// TwinCAT 3 PLC project PLC
// ProgramVersion: 3.1.4023.0
// libraries:
//   Tc2_Standard, * (Beckhoff Automation GmbH)
//   Tc2_System, * (Beckhoff Automation GmbH)
//   Tc2_Utilities, * (Beckhoff Automation GmbH)
//   Tc3_Module, * (Beckhoff Automation GmbH)
//   AX_Standard,1.24,Automate-X Ltd.
// project tree:
//   DUTs/Safety/ ST_Safety.TcDUT
//   GVLs/ GVL_EAP.TcGVL, GVL_HMI.TcGVL, GVL_IO.TcGVL, GVL_System.TcGVL, GVL_Recipe.TcGVL, GVL_Safety.TcGVL, GVL_Seq.TcGVL
//   / PlcTask.TcTTO
//   POUs/02 IO Mapping/ InputMapping.TcPOU, OutputMapping.TcPOU
//   POUs/03 Equipment/ DeviceInputs.TcPOU, DeviceOutputs.TcPOU
//   POUs/04 Program/ ExampleSequence.TcPOU
//   POUs/06 Safety/ Safety.TcPOU
//   POUs/09 General/ DataControl.TcPOU
//   POUs/10 EAP/ EAP_PublisherMapping.TcPOU, EAP_SubscriberMapping.TcPOU
//   POUs/ MachineStatePackML.TcPOU, MAIN.TcPOU
// real-time tasks:
//   TASK PlcTask: cycle T#10ms, priority 20, ADS port 350

CONFIGURATION PLC
    RESOURCE PLC ON TwinCAT3
        TASK PlcTask(INTERVAL := T#10ms, PRIORITY := 20);
        PROGRAM MAIN WITH PlcTask : MAIN;
    END_RESOURCE
END_CONFIGURATION

// ---- DUTs/Safety/ST_Safety.TcDUT
TYPE ST_Safety :
STRUCT
	

	//Basic Safety variables, add more if needed.
	bEStop					: BOOL;
	bEnergised				: BOOL;
	bHealthy				: BOOL;
	bEStopOk				: BOOL;
	bEStopResetRequired		: BOOL;
	

END_STRUCT
END_TYPE

// ---- GVLs/GVL_EAP.TcGVL
{attribute 'qualified_only'}

// Set size of array according to EAP data to be exchanged.

VAR_GLOBAL
	aPubBool		AT %Q*	: ARRAY [0..15] OF BOOL;		// EAP Published Array of Booleans
	aPubInt			AT %Q*	: ARRAY [0..15] OF INT;			// EAP Published Array of Integers
	aPubReal		AT %Q*	: ARRAY [0..15] OF REAL;		// EAP Published Array of Reals
	aSubBool		AT %I*	: ARRAY [0..15] OF BOOL;		// EAP Subscribed Array of Booleans
	aSubInt			AT %I*	: ARRAY [0..15] OF INT;			// EAP Subscribed Array of Integers
	aSubReal		AT %I*	: ARRAY [0..15] OF REAL;		// EAP Subscribed Array of Reals
END_VAR

// ---- GVLs/GVL_HMI.TcGVL
{attribute 'qualified_only'}
VAR_GLOBAL
END_VAR

// ---- GVLs/GVL_IO.TcGVL
{attribute 'qualified_only'}
VAR_GLOBAL
	

(* --- Digital Inputs --- *)


//Examples
//stPE3001				: ST_DigitalInput;
//stDI1001				: ST_DigitalInput;
//stPB4001				: ST_DigitalInput;
//stES4001				: ST_Safe2ChDigitalInput;		//PLC Cabinet Estop


(* --- Digital Outputs --- *)

//Examples
//stDO1001				: ST_DigitalOutput;		
//stDO1002				: ST_DigitalOutput;
//stSO4001				: ST_DigitalOutput;				//SO4001 Sounder


(* --- Analog Inputs --- *)

//Examples
//stAI4001				: ST_AnalogueInput;		
//stAI3001				: ST_AnalogueInput;



(* --- Analog Outputs --- *)

//Examples
//stAO4001				: ST_AnalogueInput;		
//stAO3001				: ST_AnalogueInput;



(* --- PLC IO Cards --- *)

//Examples
//stEL1008				: ST_EL1008; 
//stEL2008				: ST_EL2008;
//stEL3024				: ST_EL3024;

END_VAR

// ---- GVLs/GVL_System.TcGVL
{attribute 'qualified_only'}
VAR_GLOBAL
	
	MachineStates: ST_PackML;
	
	bResetSequenceTimerDefaults			: BOOL;				// Resets Sequence Timers to Defaults
	bSetDebounceTimes					: BOOL;				// Sets Photoeye Debounce Timers
	
END_VAR

// ---- GVLs/GVL_Recipe.TcGVL
{attribute 'qualified_only'}
VAR_GLOBAL
END_VAR

// ---- GVLs/GVL_Safety.TcGVL
{attribute 'qualified_only'}
VAR_GLOBAL
	

	stSafety			: ST_Safety;
	stSafetySeq			: ST_Sequence;
	fbSafetySeq			: FB_Sequence;
	
	bResetTrigger 		: BOOL; // from HMI or physical reset button

	bRun		AT %Q* 	: BOOL;	// To safety PLC
	bErrorAck   AT %Q* 	: BOOL;	// To safety PLC
	bReset    	AT %Q* 	: BOOL;	// To safety PLC
	
	bRunStatus  AT %I* 	: BOOL;	// From safety PLC
	
	bRequestToEnter		: BOOL; // Used with safety cages/doors
	
END_VAR

// ---- GVLs/GVL_Seq.TcGVL
{attribute 'qualified_only'}
VAR_GLOBAL
	
//List all sequencies 

//Example
//S101	 								: ST_Sequence;
//S102 									: ST_Sequence;

(* Exmaple Sequencies *)
stExampleSequence 						: ST_Sequence;
ExampleSequence_bHomingRequired 		: BOOL;

//Call  FB_Sequence for each sequence

//Example
//fbS101 								: FB_Sequence;
//fbS102 								: FB_Sequence;

(* Exmaple FB *)
fbExampleSequence : FB_Sequence;

// When used with conveyors , additions to Sequencies have been used on previous projects such as:
//S101_RequestingToSend		: BOOL;
//S101_ReadyToReceive       : BOOL; 

// When used with moving parts , additions to Sequencies have been used on previous projects such as:
//S101_bHomingRequired 		: BOOL;

END_VAR

// ---- POUs/MAIN.TcPOU
PROGRAM MAIN
VAR
END_VAR


// Add and Call Programs to be used 

//	InputMapping();
//	DeviceInputs();
//	Seq1();
//	Safety();
//	MachineStatePackML();
//	DataControl();
//	OutputMapping();
//	DeviceOutputs();
//	EAP_SubscriberMapping();
//	EAP_PublisherMapping();

END_PROGRAM

// ---- POUs/06 Safety/Safety.TcPOU
PROGRAM Safety
VAR
END_VAR


// Call Safety Sequence Function Block
GVL_Safety.fbSafetySeq(stSeq:=GVL_Safety.stSafetySeq);


CASE GVL_Safety.stSafetySeq.nStep OF
	0:	// Aborted
		// Actions
		
		
		// Step Transitions
		IF (GVL_Safety.bResetTrigger AND GVL_Safety.stSafetySeq.bStepTimerDn) THEN
			GVL_Safety.stSafetySeq.nNewStep := 1;
		END_IF
		
	1:	// Safety Reset Step 1
		// Actions
		
		// Step Transitions
		IF GVL_Safety.stSafetySeq.bStepTimerDn THEN
			GVL_Safety.stSafetySeq.nNewStep := 2;
		END_IF 
		
	2:	// Safety Reset Step 2
		// Actions

		// Step Transitions
		IF GVL_Safety.stSafetySeq.bStepTimerDn THEN
			GVL_Safety.stSafetySeq.nNewStep := 3;
		END_IF
		
	3:	// Safety Reset Step 3
		// Actions

		// Step Transitions
		IF GVL_Safety.stSafetySeq.bStepTimerDn AND GVL_Safety.stSafety.bHealthy THEN
			
			GVL_Safety.stSafetySeq.nNewStep := 4;
		END_IF 
		
	4: //System Reset Step 1
		// Actions
			
		// Step Transitions
		IF GVL_Safety.stSafetySeq.bStepTimerDn THEN
			GVL_Safety.stSafetySeq.nNewStep := 5;
		END_IF 

	5:	//System Reset Step 2
		// Actions

		// Step Transitions
		IF GVL_Safety.stSafetySeq.bStepTimerDn THEN
			GVL_Safety.stSafetySeq.nNewStep := 6;
		END_IF
		
	6: 	//System Reset Complete
		//Actions
		
		//Step Transitions

	
END_CASE

IF GVL_Safety.bResetTrigger THEN
	GVL_Safety.stSafetySeq.nNewStep := 1;
END_IF  

IF NOT GVL_Safety.stSafety.bHealthy THEN
	GVL_Safety.stSafetySeq.nNewStep := 0;
END_IF	

WriteToFlags();
WriteToOutputs();

ACTION WriteToFlags:




//Safety Group Run
IF 	GVL_Safety.stSafetySeq.nStep = 1 OR
	GVL_Safety.stSafetySeq.nStep = 2 OR
	GVL_Safety.stSafetySeq.nStep = 3 OR
	GVL_Safety.stSafetySeq.nStep = 4 OR
	GVL_Safety.stSafetySeq.nStep = 5 OR
	GVL_Safety.stSafetySeq.nStep = 6
THEN
	GVL_Safety.bRun := TRUE;
ELSE
	GVL_Safety.bRun := FALSE;
END_IF
		
//Safety Group Error Acknowledge Reset
IF 
	GVL_Safety.stSafetySeq.nStep = 2
THEN
	GVL_Safety.bErrorAck := TRUE;
ELSE
	GVL_Safety.bErrorAck := FALSE;
END_IF			
		

//Safety Function Block Resets
IF 
	GVL_Safety.stSafetySeq.nStep = 2
THEN
	GVL_Safety.bReset := TRUE;
ELSE
	GVL_Safety.bReset := FALSE;
END_IF
END_ACTION

ACTION WriteToOutputs:

END_ACTION

END_PROGRAM

// ---- POUs/02 IO Mapping/InputMapping.TcPOU
(*****************************************************************************************
	Automate-X Ltd. © 
	www.automate-x.nz 	
	
	Map Physical Inputs to device structures
******************************************************************************************)

PROGRAM InputMapping
VAR
END_VAR



// Map physical inputs (based on PLC IO Cards in GVL IO) to device structures
// This is IO Assignment based on PLC IO List in Equipment schedule



// This EXAMPLE is based on variables in GVL_IO

//EL1008 | 8-channel digital input terminal 24 V DC, 3 ms

//GVL_IO.stPE3001.bInput		:=  GVL_IO.stEL1008.bDI1;
//GVL_IO.stDI1001.bInput		:=  GVL_IO.stEL1008.bDI2;
//GVL_IO.stPB4001.bInput		:=  GVL_IO.stEL1008.bDI3;
// SPARE            		:=  GVL_IO.stEL1008.bDI4;
// SPARE            		:=  GVL_IO.stEL1008.bDI5;
// SPARE            		:=  GVL_IO.stEL1008.bDI6;
// SPARE            		:=  GVL_IO.stEL1008.bDI7;
// SPARE            		:=  GVL_IO.stEL1008.bDI8;



//EL3024 | 4-channel Analog Input terminal ,Current , 4..20mA, 12bit, Differential

//GVL_IO.stAO4001.bInput		:=  GVL_IO.stEL3024.bAI1;
//GVL_IO.stAO3001.bInput		:=  GVL_IO.stEL3024.bAI2;
// SPARE  					:=  GVL_IO.stEL3024.bAI3;
// SPARE            		:=  GVL_IO.stEL3024.bAI4;

END_PROGRAM

// ---- POUs/02 IO Mapping/OutputMapping.TcPOU
(*****************************************************************************************
	Automate-X Ltd. © 
	www.automate-x.nz 	
	
	Map Physical Outputs to device structures
******************************************************************************************)


PROGRAM OutputMapping
VAR
END_VAR




// Map physical inputs (based on PLC IO Cards in GVL IO) to device structures
// This is IO Assignment based on PLC IO List in Equipment schedule



// This EXAMPLE is based on variables in GVL_IO

//EL2008 | 8-channel digital Output terminal 24 V DC, 3 ms

//GVL_IO.stDO1001.bOutput		:=  GVL_IO.stEL2008.bDO1;
//GVL_IO.stDO1002.bOutput		:=  GVL_IO.stEL2008.bDO2;
//GVL_IO.stSO4001.bOutput		:=  GVL_IO.stEL2008.bDO3;
// SPARE            		:=  GVL_IO.stEL2008.bDO4;
// SPARE            		:=  GVL_IO.stEL2008.bDO5;
// SPARE            		:=  GVL_IO.stEL2008.bDO6;
// SPARE            		:=  GVL_IO.stEL2008.bDO7;
// SPARE            		:=  GVL_IO.stEL2008.bDO8;

END_PROGRAM

// ---- POUs/03 Equipment/DeviceInputs.TcPOU
(*****************************************************************************************
	Automate-X Ltd. ©  
	www.automate-x.nz 	
	
	Initialise and call all function blocks for Input type devices
******************************************************************************************)

PROGRAM DeviceInputs
VAR
	
//Example 
// fbPX01    	: FB_DigitalInput;
// fbDI1002		: FB_DigitalInput;		
// fbPE3001		: FB_DigitalInput;

END_VAR



// Call Function Block instances and use defined data type for the input device

//Example
//fbPE3001(	stDI	:= GVL_IO.stPE3001);
//fbDI1001(	stDI 	:= GVL_IO.stDI1001);			
//fbPB4001(	stDI 	:= GVL_IO.stPB4001);

END_PROGRAM

// ---- POUs/03 Equipment/DeviceOutputs.TcPOU
(*****************************************************************************************
	Automate-X Ltd. © 
	www.automate-x.nz 	
	
	Initialise and call all function blocks for Output type devices
******************************************************************************************)

PROGRAM DeviceOutputs
VAR
	
//Example
//fbDO1001	: FB_DigitalOutput;		
//fbDO1002	: FB_DigitalOutput;    


END_VAR


// Call Function Block instances and use defined data type for the input device

//Example
//fbDO1001(stDQ := GVL_IO.stDO1001);		
//fbDO1002(stDQ := GVL_IO.stDO1002);

END_PROGRAM

// ---- POUs/04 Program/ExampleSequence.TcPOU
PROGRAM ExampleSequence
VAR
END_VAR



// Call Sequence Function Block
GVL_Seq.fbExampleSequence(stSeq:=GVL_Seq.stExampleSequence);
GVL_Seq.stExampleSequence.sSeqName := 'Example Sequence';
GVL_Seq.stExampleSequence.sSeqDesc := 'stExampleSequence - Example Sequence';


(* Insert sequence based on Grafcet FD *)
(* Changes to the sequence must be done in the FD first, then code changes can be implemented *)
(* Add & modify steps as necessary *)

CASE GVL_Seq.stExampleSequence.nStep OF
	
	0:	// Aborted
		// Message
		GVL_Seq.stExampleSequence.sSeqMsg := 'Aborted';
			
		// Step Transitions		
	
	1:	// Idle
		// Message
		GVL_Seq.stExampleSequence.sSeqMsg := 'Idle';
		
		
		// Step Transitions
		
			
	2:	// Fault
		// Message
		GVL_Seq.stExampleSequence.sSeqMsg := 'Fault';
		
		// Step Transitions
		
			
	4:	// Held
		// Message
		GVL_Seq.stExampleSequence.sSeqMsg := 'Held';
		
		// Step Transitions
		
		

	5:	// Check State
		// Message
		GVL_Seq.stExampleSequence.sSeqMsg := 'Check State';
		

		// Step Transitions
		
	
	6: // Home System
		// Message
		GVL_Seq.stExampleSequence.sSeqMsg := 'Home System';
		
		// Step Transitions
		

	7: // 
		// Message
		GVL_Seq.stExampleSequence.sSeqMsg := '';
		
		// Step Transitions
		
		
	8: // 
		// Message
		GVL_Seq.stExampleSequence.sSeqMsg := '';
		
		// Step Transitions
		
	9: // 
		// Message
		GVL_Seq.stExampleSequence.sSeqMsg := '';
		
		// Step Transitions
		
	10: // 
		// Message
		GVL_Seq.stExampleSequence.sSeqMsg := '';
		
		// Step Transitions
	
		
END_CASE

WriteToOutputs();
WriteToFlags();

ACTION WriteToFlags:


(* Flags Setting and Resetting is determined by the sequence matrix in the Grafcet FD *)


//		IF 		GVL_Seq.stExampleSequence.nNewStep 		= 7
//			OR 	GVL_Seq.stExampleSequence.nNewStep 		= 8
//			OR 	GVL_Seq.stExampleSequence.nNewStep 		= 9
//			OR 	GVL_Seq.stExampleSequence.nNewStep 		= 10
//		THEN
//			ADD Flag Here := TRUE;
//		ELSE
//			ADD Flag Here := FALSE;
//		END_IF
END_ACTION

ACTION WriteToOutputs:



(* Outputs Setting and Resetting is determined by the sequence matrix in the Grafcet FD *)

//		IF 		GVL_Seq.stExampleSequence.nNewStep 		= 7
//			OR 	GVL_Seq.stExampleSequence.nNewStep 		= 8
//			OR 	GVL_Seq.stExampleSequence.nNewStep 		= 9
//			OR 	GVL_Seq.stExampleSequence.nNewStep 		= 10
//		THEN
//			ADD Output Here := TRUE;
//		ELSE
//			ADD Output Here := FALSE;
//		END_IF
END_ACTION

END_PROGRAM

// ---- POUs/09 General/DataControl.TcPOU
PROGRAM DataControl
VAR
	
END_VAR



// Use what's needed and delete unused methods

// IF GVL_System.bResetSequenceTimerDefaults 	THEN
// 	M_ResetSequenceTimerDefaults();
// 	GVL_System.bResetSequenceTimerDefaults	:= FALSE;
// END_IF


// IF GVL_System.bSetDebounceTimes 	THEN
// 	M_SetDebounceTimes();
// 	GVL_System.bSetDebounceTimes	:= FALSE;
// END_IF


//M_WritePersistentData();


// Use this method to set Steptimes for sequence steps 
// This is copied from Steptimers tab in the Grafcet FD

METHOD M_ResetSequenceTimerDefaults : BOOL
VAR_INPUT
END_VAR

// Example

// GVL_Safety.stSafetySeq.aStepTimes[0] := T#300MS;
// GVL_Safety.stSafetySeq.aStepTimes[1] := T#300MS;
// GVL_Safety.stSafetySeq.aStepTimes[2] := T#300MS;
// GVL_Safety.stSafetySeq.aStepTimes[3] := T#300MS;
// GVL_Safety.stSafetySeq.aStepTimes[4] := T#300MS;
// GVL_Safety.stSafetySeq.aStepTimes[5] := T#300MS;

// GVL_Seq.stExampleSequence.aStepTimes[0] := T#0MS;
// GVL_Seq.stExampleSequence.aStepTimes[1] := T#0MS;
// GVL_Seq.stExampleSequence.aStepTimes[2] := T#0MS;
// GVL_Seq.stExampleSequence.aStepTimes[3] := T#0MS;
// GVL_Seq.stExampleSequence.aStepTimes[4] := T#0MS;
// GVL_Seq.stExampleSequence.aStepTimes[5] := T#500MS;
// GVL_Seq.stExampleSequence.aStepTimes[6] := T#0MS;
// GVL_Seq.stExampleSequence.aStepTimes[7] := T#0MS;
// GVL_Seq.stExampleSequence.aStepTimes[8] := T#0MS;
// GVL_Seq.stExampleSequence.aStepTimes[9] := T#0MS;
// GVL_Seq.stExampleSequence.aStepTimes[10] := T#0MS;
END_METHOD


// Use this method to set debounce timers on I/O
METHOD M_SetDebounceTimes : BOOL
VAR_INPUT
END_VAR

// Example

//GVL_IO.PE101.tDebounceOff_PT	:= T#100MS;
//GVL_IO.PE103.tDebounceOn_PT	:= T#250MS;
END_METHOD


//To be Used only if IPC has 1-second UPS (for example: CX9020)
// If not needed, delete from Project 

METHOD M_WritePersistentData : BOOL
VAR_INPUT
END_VAR
VAR
	FB_WritePersistentData		: FB_WritePersistentData;
	RT_WritePersistent			: R_TRIG;
	bWritePersistent			: BOOl;
END_VAR


RT_WritePersistent(CLK:=bWritePersistent);
FB_WritePersistentData(NETID:='', PORT:=851, START:= RT_WritePersistent.Q, TMOUT:=T#1S );
bWritePersistent	:= FALSE;
END_METHOD

END_PROGRAM

// ---- POUs/10 EAP/EAP_PublisherMapping.TcPOU
(*****************************************************************************************
	Automate-X Ltd. © 2020 
	www.automate-x.nz 	
	
	Map out EAP (EtherCAT Automation Protocol) Publisher Variables.
	This is done instead of direct subscribing due to limitations around custom DUTs in libraries.
******************************************************************************************)
PROGRAM EAP_PublisherMapping
VAR
END_VAR


//Add or remove data points according to size of arrays in GVL_EAP

//GVL_EAP.aPubBool[0] :=;
//GVL_EAP.aPubBool[1] :=;
//GVL_EAP.aPubBool[2] :=;
//GVL_EAP.aPubBool[3] :=;
//GVL_EAP.aPubBool[4] :=;
//GVL_EAP.aPubBool[5] :=;
//GVL_EAP.aPubBool[6] :=;
//GVL_EAP.aPubBool[7] :=;
//GVL_EAP.aPubBool[8] :=;
//GVL_EAP.aPubBool[9] :=;
//GVL_EAP.aPubBool[10] :=;
//GVL_EAP.aPubBool[11] :=;
//GVL_EAP.aPubBool[12] := ;
//GVL_EAP.aPubBool[13] := ;
//GVL_EAP.aPubBool[14] := ;
//GVL_EAP.aPubBool[15] := ;
//GVL_EAP.aPubBool[16] := ;


//GVL_EAP.aPubInt[0] := ;
//GVL_EAP.aPubInt[1] := ;
//GVL_EAP.aPubInt[2] := ;
//GVL_EAP.aPubInt[3] := ;
//GVL_EAP.aPubInt[4] := ;
//GVL_EAP.aPubInt[5] := ;
//GVL_EAP.aPubInt[6] := ;
//GVL_EAP.aPubInt[7] := ;
//GVL_EAP.aPubInt[8] := ;
//GVL_EAP.aPubInt[9] := ;
//GVL_EAP.aPubInt[10] := ;
//GVL_EAP.aPubInt[11] := ;
//GVL_EAP.aPubInt[12] := ;
//GVL_EAP.aPubInt[13] := ;
//GVL_EAP.aPubInt[14] := ;
//GVL_EAP.aPubInt[15] := ;

//GVL_EAP.aPubReal[0] := ;
//GVL_EAP.aPubReal[1] := ;
//GVL_EAP.aPubReal[2] := ;
//GVL_EAP.aPubReal[3] := ;
//GVL_EAP.aPubReal[4] := ;
//GVL_EAP.aPubReal[5] := ;
//GVL_EAP.aPubReal[6] := ;
//GVL_EAP.aPubReal[7] := ;
//GVL_EAP.aPubReal[8] := ;
//GVL_EAP.aPubReal[9] := ;
//GVL_EAP.aPubReal[10] := ;
//GVL_EAP.aPubReal[11] := ;
//GVL_EAP.aPubReal[12] := ;
//GVL_EAP.aPubReal[13] := ;
//GVL_EAP.aPubReal[14] := ;
//GVL_EAP.aPubReal[15] := ;

END_PROGRAM

// ---- POUs/10 EAP/EAP_SubscriberMapping.TcPOU
(*****************************************************************************************
	Automate-X Ltd. © 2020 
	www.automate-x.nz 	
	
	Map in EAP (EtherCAT Automation Protocol) Subscriber Variables.
	This is done instead of direct subscribing due to limitations around custom DUTs in libraries.
******************************************************************************************)
PROGRAM EAP_SubscriberMapping
VAR
END_VAR


//Add or remove data points according to size of arrays in GVL_EAP

//GVL_EAP.aSubBool[0] :=;
//GVL_EAP.aSubBool[1] :=;
//GVL_EAP.aSubBool[2] :=;
//GVL_EAP.aSubBool[3] :=;
//GVL_EAP.aSubBool[4] :=;
//GVL_EAP.aSubBool[5] :=;
//GVL_EAP.aSubBool[6] :=;
//GVL_EAP.aSubBool[7] :=;
//GVL_EAP.aSubBool[8] :=;
//GVL_EAP.aSubBool[9] :=;
//GVL_EAP.aSubBool[10] :=;
//GVL_EAP.aSubBool[11] :=;
//GVL_EAP.aSubBool[12] := ;
//GVL_EAP.aSubBool[13] := ;
//GVL_EAP.aSubBool[14] := ;
//GVL_EAP.aSubBool[15] := ;
//GVL_EAP.aSubBool[16] := ;

//GVL_EAP.aSubInt[0] := ;
//GVL_EAP.aSubInt[1] := ;
//GVL_EAP.aSubInt[2] := ;
//GVL_EAP.aSubInt[3] := ;
//GVL_EAP.aSubInt[4] := ;
//GVL_EAP.aSubInt[5] := ;
//GVL_EAP.aSubInt[6] := ;
//GVL_EAP.aSubInt[7] := ;
//GVL_EAP.aSubInt[8] := ;
//GVL_EAP.aSubInt[9] := ;
//GVL_EAP.aSubInt[10] := ;
//GVL_EAP.aSubInt[11] := ;
//GVL_EAP.aSubInt[12] := ;
//GVL_EAP.aSubInt[13] := ;
//GVL_EAP.aSubInt[14] := ;
//GVL_EAP.aSubInt[15] := ;

//GVL_EAP.aSubReal[0] := ;
//GVL_EAP.aSubReal[1] := ;
//GVL_EAP.aSubReal[2] := ;
//GVL_EAP.aSubReal[3] := ;
//GVL_EAP.aSubReal[4] := ;
//GVL_EAP.aSubReal[5] := ;
//GVL_EAP.aSubReal[6] := ;
//GVL_EAP.aSubReal[7] := ;
//GVL_EAP.aSubReal[8] := ;
//GVL_EAP.aSubReal[9] := ;
//GVL_EAP.aSubReal[10] := ;
//GVL_EAP.aSubReal[11] := ;
//GVL_EAP.aSubReal[12] := ;
//GVL_EAP.aSubReal[13] := ;
//GVL_EAP.aSubReal[14] := ;
//GVL_EAP.aSubReal[15] := ;

END_PROGRAM

// ---- POUs/MachineStatePackML.TcPOU
PROGRAM MachineStatePackML
VAR
	
 //MachineStateCurrent	: INT;
 machineState			: FB_PackML;
tonStopRequest	: TON;
(*	Aborted		:= 0,
	Aborting	:= 1,
	
	Clearing	:= 2,
	Stopping	:= 3,
	Stopped		:= 4,
	
	Resetting	:= 5,
	Idle		:= 6,
	
	Starting	:= 7,
	Execute		:= 8,
	
	Holding		:= 9,
	Unholding	:= 10,
	Held		:= 11,
	
	Completing	:= 12,
	Complete	:= 13
	
*)
	
	
END_VAR


// Conditions are just an exmaple; modify as per application requirements.


// Machine state
machineState(stPackML := GVL_System.MachineStates);


// Abort - (Abort Conditions eg EStop pressed)
GVL_System.MachineStates.bAbort := (NOT GVL_Safety.stSafety.bEStopOk AND NOT GVL_Safety.stSafety.bEStopResetRequired);
								  
// Clear - (Clear Conditions eg EStop Healthy)
GVL_System.MachineStates.bClear := GVL_Safety.stSafety.bEStopOk;

// Stop - (Stop conditions eg Stop Button)
GVL_System.MachineStates.bStop := tonStopRequest.Q;

// Reset - Reset button
GVL_System.MachineStates.bReset := GVL_Safety.bResetTrigger; 

// Start - Start button
GVL_System.MachineStates.bStart := GVL_Safety.stSafety.bEStopOk; 

// Hold - (Hold Conditions eg Request to Enter PB on a safety door/cage)

GVL_System.MachineStates.bHold := GVL_Safety.bRequestToEnter;

// Unhold - (UnHold Conditions eg Reset Trigger)
GVL_System.MachineStates.bUnhold := GVL_Safety.bResetTrigger;

// Holding - From Sequences
GVL_System.MachineStates.bHoldingSC := GVL_Seq.stExampleSequence.bHeld ;


//////////////////////////////////////////////////////////////////////////////////
// Other Conditions (Delete if not used)

// Homing Required conditions
IF GVL_System.MachineStates.bClearing (*  AND Other conditions *) THEN
	GVL_Seq.ExampleSequence_bHomingRequired := TRUE;
END_IF
	
// Stop the machine if a hold is requested but not achieved within 10s
tonStopRequest(IN:=(GVL_System.MachineStates.bHold AND NOT GVL_System.MachineStates.bHeld), PT:=T#10S);

//////////////////////////////////////////////////////////////////////////////////


// Unconditional
GVL_System.MachineStates.bAbortingSC 	:= TRUE;
GVL_System.MachineStates.bClearingSC 	:= TRUE;
GVL_System.MachineStates.bStoppingSC 	:= TRUE;
GVL_System.MachineStates.bResettingSC	:= TRUE;
GVL_System.MachineStates.bStartingSC 	:= TRUE;
GVL_System.MachineStates.bUnholdingSC := TRUE;

END_PROGRAM
